(* Logix 5000 project; controller Generic 1768-L43 rev 15.6; software revision 15.01; part 10 of 10 *)
(* tags used below, declared in another part *)
   Axis_00_CMD : UDT_Axis_CMD;
   Axis_00_Data : UDT_Axis_Data;
   AXIS_01 : AXIS_SERVO_DRIVE;
   Axis_01_CMD : UDT_Axis_CMD;
   Axis_01_Data : UDT_Axis_Data;
   Axis_01_Status : UDT_Axis_Status;
   AXIS_02 : AXIS_SERVO_DRIVE;
   Axis_02_CMD : UDT_Axis_CMD;
   Axis_02_Data : UDT_Axis_Data;
   Axis_02_Status : UDT_Axis_Status;
   AXIS_03 : AXIS_SERVO_DRIVE;
   Axis_03_CMD : UDT_Axis_CMD;
   Axis_03_Data : UDT_Axis_Data;
   Axis_03_Status : UDT_Axis_Status;
   AXIS_04 : AXIS_SERVO_DRIVE;
   Axis_04_CMD : UDT_Axis_CMD;
   Axis_04_Data : UDT_Axis_Data;
   Axis_04_Status : UDT_Axis_Status;
   GenericMachine_COND : UDT_Machine_COND;
   GUI_Axis_01_JogFwdREQ : BOOL;
   GUI_Axis_01_JogRevREQ : BOOL;
   GUI_Axis_01_ReferenceREQ : BOOL;
   GUI_Axis_02_JogFwdREQ : BOOL;
   GUI_Axis_02_JogRevREQ : BOOL;
   GUI_Axis_02_ReferenceREQ : BOOL;
   GUI_Axis_03_JogFwdREQ : BOOL;
   GUI_Axis_03_JogRevREQ : BOOL;
   GUI_Axis_03_ReferenceREQ : BOOL;
   GUI_Axis_04_JogFwdREQ : BOOL;
   GUI_Axis_04_JogRevREQ : BOOL;
   GUI_Axis_04_ReferenceREQ : BOOL;
   GUI_ReferenceREQ : BOOL;
   PhaseTimout : UDT_PhaseTimeout;
   PZ_GenericMachine_AUTO : PHASE;
   PZ_GenericMachine_MANUAL : PHASE;
(* PZ_GenericMachine_AUTO, continued *)

ROUTINE Running   (* ladder *)
// CONTROLS MACHINE RUNNING PHASE.  MODIFY AS NEEDED.
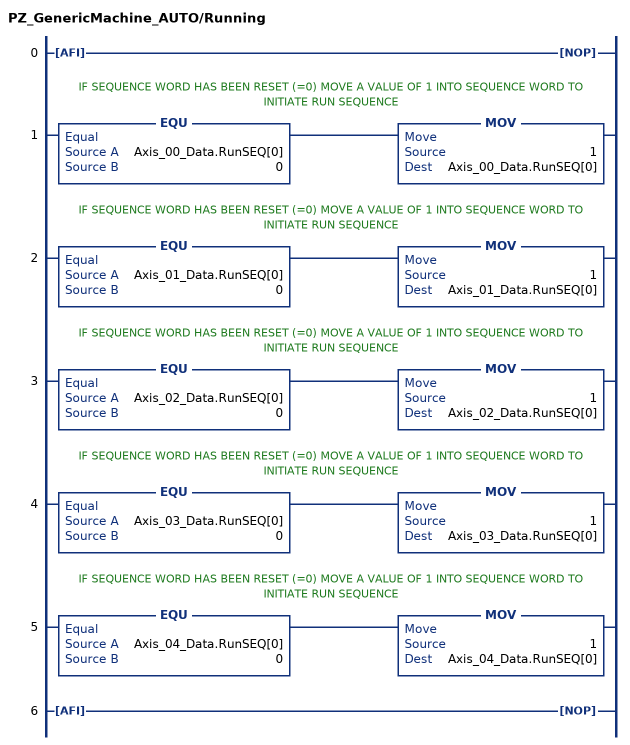
   0: AFI()NOP();
   // IF SEQUENCE WORD HAS BEEN RESET (=0) MOVE A VALUE OF 1 INTO SEQUENCE WORD TO INITIATE RUN SEQUENCE
   1: EQU(Axis_00_Data.RunSEQ[0],0)MOV(1,Axis_00_Data.RunSEQ[0]);
   // IF SEQUENCE WORD HAS BEEN RESET (=0) MOVE A VALUE OF 1 INTO SEQUENCE WORD TO INITIATE RUN SEQUENCE
   2: EQU(Axis_01_Data.RunSEQ[0],0)MOV(1,Axis_01_Data.RunSEQ[0]);
   // IF SEQUENCE WORD HAS BEEN RESET (=0) MOVE A VALUE OF 1 INTO SEQUENCE WORD TO INITIATE RUN SEQUENCE
   3: EQU(Axis_02_Data.RunSEQ[0],0)MOV(1,Axis_02_Data.RunSEQ[0]);
   // IF SEQUENCE WORD HAS BEEN RESET (=0) MOVE A VALUE OF 1 INTO SEQUENCE WORD TO INITIATE RUN SEQUENCE
   4: EQU(Axis_03_Data.RunSEQ[0],0)MOV(1,Axis_03_Data.RunSEQ[0]);
   // IF SEQUENCE WORD HAS BEEN RESET (=0) MOVE A VALUE OF 1 INTO SEQUENCE WORD TO INITIATE RUN SEQUENCE
   5: EQU(Axis_04_Data.RunSEQ[0],0)MOV(1,Axis_04_Data.RunSEQ[0]);
   6: AFI()NOP();
END_ROUTINE

ROUTINE Stopping   (* ladder *)
// CONTROLS MACHINE STOPPING PHASE.  MODIFY AS NEEDED.
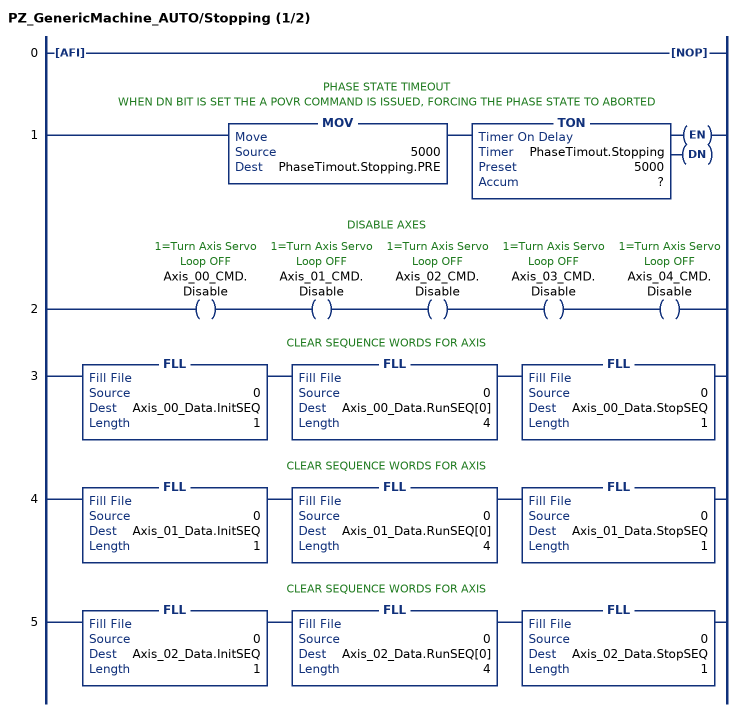
   0: AFI()NOP();
   // PHASE STATE TIMEOUT
   //   WHEN DN BIT IS SET THE A POVR COMMAND IS ISSUED, FORCING THE PHASE STATE TO ABORTED
   1: MOV(5000,PhaseTimout.Stopping.PRE)TON(PhaseTimout.Stopping,?,?);
   // DISABLE AXES
   2: OTE(Axis_00_CMD.Disable)OTE(Axis_01_CMD.Disable)OTE(Axis_02_CMD.Disable)OTE(Axis_03_CMD.Disable)OTE(Axis_04_CMD.Disable);
   // CLEAR SEQUENCE WORDS FOR AXIS
   3: FLL(0,Axis_00_Data.InitSEQ,1)FLL(0,Axis_00_Data.RunSEQ[0],4)FLL(0,Axis_00_Data.StopSEQ,1);
   // CLEAR SEQUENCE WORDS FOR AXIS
   4: FLL(0,Axis_01_Data.InitSEQ,1)FLL(0,Axis_01_Data.RunSEQ[0],4)FLL(0,Axis_01_Data.StopSEQ,1);
   // CLEAR SEQUENCE WORDS FOR AXIS
   5: FLL(0,Axis_02_Data.InitSEQ,1)FLL(0,Axis_02_Data.RunSEQ[0],4)FLL(0,Axis_02_Data.StopSEQ,1);
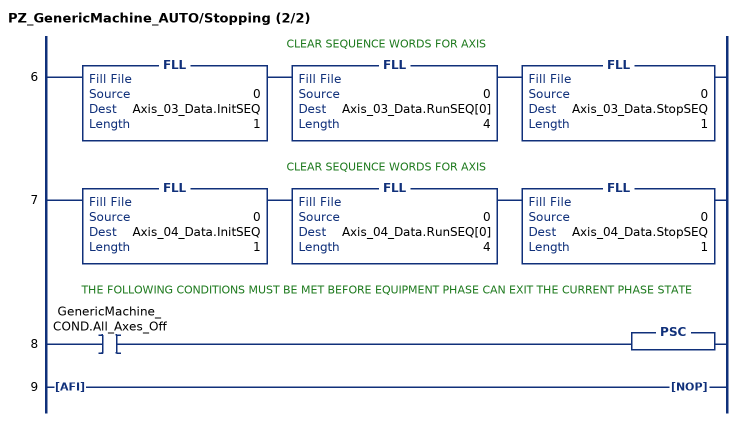
   // CLEAR SEQUENCE WORDS FOR AXIS
   6: FLL(0,Axis_03_Data.InitSEQ,1)FLL(0,Axis_03_Data.RunSEQ[0],4)FLL(0,Axis_03_Data.StopSEQ,1);
   // CLEAR SEQUENCE WORDS FOR AXIS
   7: FLL(0,Axis_04_Data.InitSEQ,1)FLL(0,Axis_04_Data.RunSEQ[0],4)FLL(0,Axis_04_Data.StopSEQ,1);
   // THE FOLLOWING CONDITIONS MUST BE MET BEFORE EQUIPMENT PHASE CAN EXIT THE CURRENT PHASE STATE
   8: XIC(GenericMachine_COND.All_Axes_Off)PSC();
   9: AFI()NOP();
END_ROUTINE
END_PROGRAM

PROGRAM PZ_GenericMachine_MANUAL

ROUTINE Aborting   (* ladder *)
// CONTROLS MACHINE MANUAL ABORTING PHASE.  MODIFY AS NEEDED.
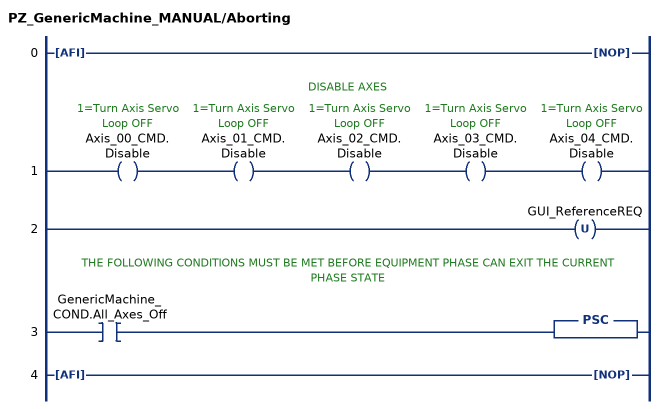
   0: AFI()NOP();
   // DISABLE AXES
   1: OTE(Axis_00_CMD.Disable)OTE(Axis_01_CMD.Disable)OTE(Axis_02_CMD.Disable)OTE(Axis_03_CMD.Disable)OTE(Axis_04_CMD.Disable);
   2: OTU(GUI_ReferenceREQ);
   // THE FOLLOWING CONDITIONS MUST BE MET BEFORE EQUIPMENT PHASE CAN EXIT THE CURRENT PHASE STATE
   3: XIC(GenericMachine_COND.All_Axes_Off)PSC();
   4: AFI()NOP();
END_ROUTINE

ROUTINE Resetting   (* ladder *)
// CONTROLS MACHINE MANUAL RESETTING PHASE.  MODIFY AS NEEDED.
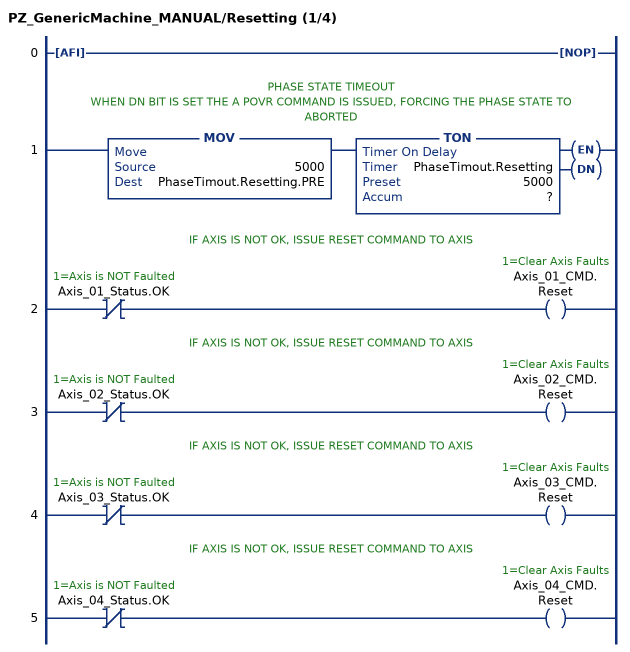
   0: AFI()NOP();
   // PHASE STATE TIMEOUT
   //   WHEN DN BIT IS SET THE A POVR COMMAND IS ISSUED, FORCING THE PHASE STATE TO ABORTED
   1: MOV(5000,PhaseTimout.Resetting.PRE)TON(PhaseTimout.Resetting,?,?);
   // IF AXIS IS NOT OK, ISSUE RESET COMMAND TO AXIS
   2: XIO(Axis_01_Status.OK)OTE(Axis_01_CMD.Reset);
   // IF AXIS IS NOT OK, ISSUE RESET COMMAND TO AXIS
   3: XIO(Axis_02_Status.OK)OTE(Axis_02_CMD.Reset);
   // IF AXIS IS NOT OK, ISSUE RESET COMMAND TO AXIS
   4: XIO(Axis_03_Status.OK)OTE(Axis_03_CMD.Reset);
   // IF AXIS IS NOT OK, ISSUE RESET COMMAND TO AXIS
   5: XIO(Axis_04_Status.OK)OTE(Axis_04_CMD.Reset);
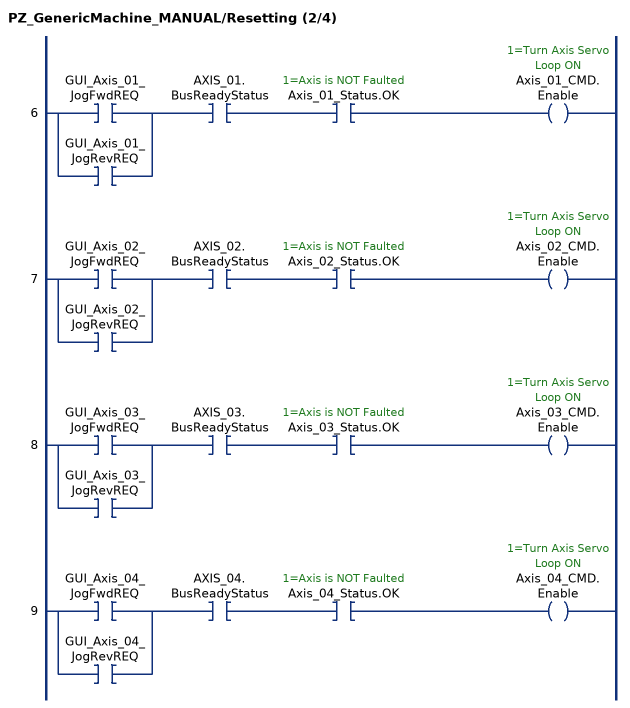
   6: [XIC(GUI_Axis_01_JogFwdREQ) ,XIC(GUI_Axis_01_JogRevREQ) ]XIC(AXIS_01.BusReadyStatus)XIC(Axis_01_Status.OK)OTE(Axis_01_CMD.Enable);
   7: [XIC(GUI_Axis_02_JogFwdREQ) ,XIC(GUI_Axis_02_JogRevREQ) ]XIC(AXIS_02.BusReadyStatus)XIC(Axis_02_Status.OK)OTE(Axis_02_CMD.Enable);
   8: [XIC(GUI_Axis_03_JogFwdREQ) ,XIC(GUI_Axis_03_JogRevREQ) ]XIC(AXIS_03.BusReadyStatus)XIC(Axis_03_Status.OK)OTE(Axis_03_CMD.Enable);
   9: [XIC(GUI_Axis_04_JogFwdREQ) ,XIC(GUI_Axis_04_JogRevREQ) ]XIC(AXIS_04.BusReadyStatus)XIC(Axis_04_Status.OK)OTE(Axis_04_CMD.Enable);
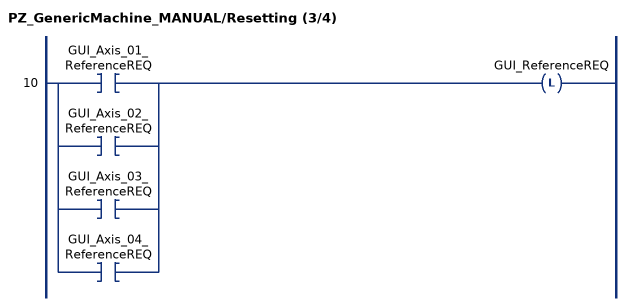
   10: [XIC(GUI_Axis_01_ReferenceREQ) ,XIC(GUI_Axis_02_ReferenceREQ) ,XIC(GUI_Axis_03_ReferenceREQ) ,XIC(GUI_Axis_04_ReferenceREQ) ]OTL(GUI_ReferenceREQ);
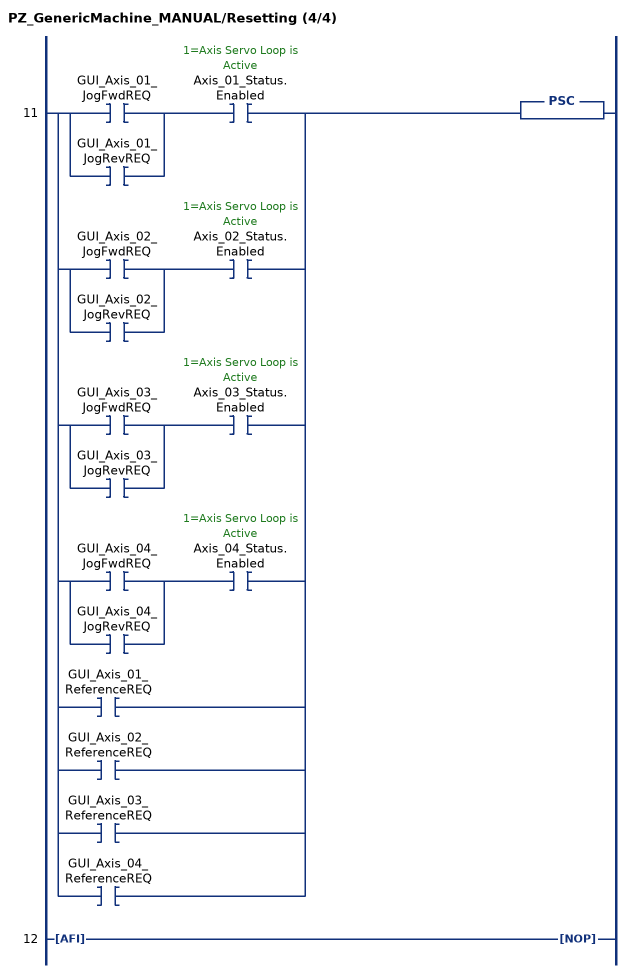
   11: [[XIC(GUI_Axis_01_JogFwdREQ) ,XIC(GUI_Axis_01_JogRevREQ) ] XIC(Axis_01_Status.Enabled) ,[XIC(GUI_Axis_02_JogFwdREQ) ,XIC(GUI_Axis_02_JogRevREQ) ] XIC(Axis_02_Status.Enabled) ,[XIC(GUI_Axis_03_JogFwdREQ) ,XIC(GUI_Axis_03_JogRevREQ) ] XIC(Axis_03_Status.Enabled) ,[XIC(GUI_Axis_04_JogFwdREQ) ,XIC(GUI_Axis_04_JogRevREQ) ] XIC(Axis_04_Status.Enabled) ,XIC(GUI_Axis_01_ReferenceREQ) ,XIC(GUI_Axis_02_ReferenceREQ) ,XIC(GUI_Axis_03_ReferenceREQ) ,XIC(GUI_Axis_04_ReferenceREQ) ]PSC();
   12: AFI()NOP();
END_ROUTINE

ROUTINE Running   (* ladder *)
// CONTROLS MACHINE MANUAL RUNNING PHASE.  MODIFY AS NEEDED.
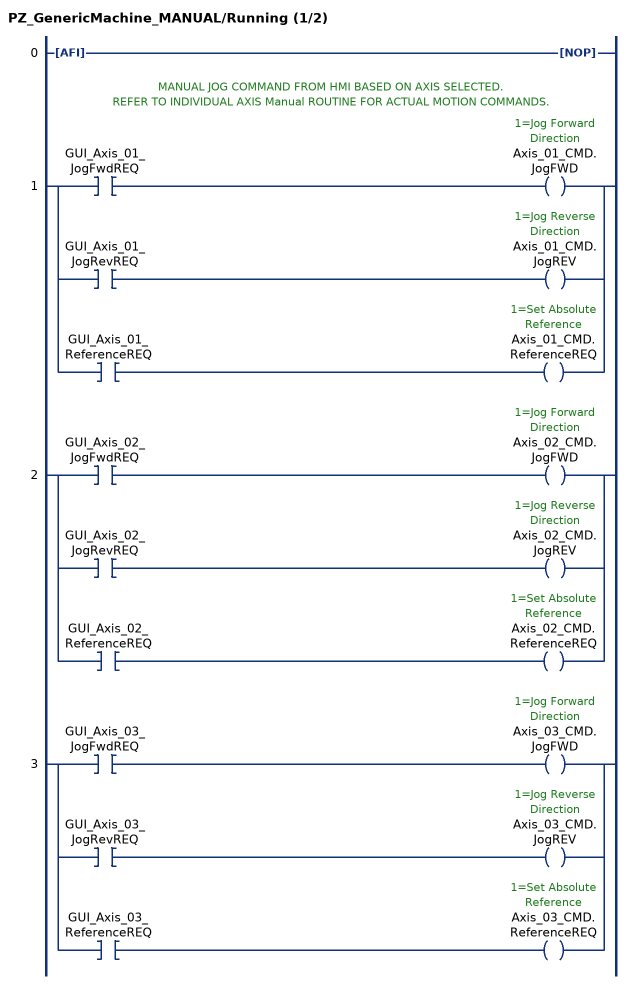
   0: AFI()NOP();
   // MANUAL JOG COMMAND FROM HMI BASED ON AXIS SELECTED.
   // REFER TO INDIVIDUAL AXIS Manual ROUTINE FOR ACTUAL MOTION COMMANDS.
   1: [XIC(GUI_Axis_01_JogFwdREQ) OTE(Axis_01_CMD.JogFWD) ,XIC(GUI_Axis_01_JogRevREQ) OTE(Axis_01_CMD.JogREV) ,XIC(GUI_Axis_01_ReferenceREQ) OTE(Axis_01_CMD.ReferenceREQ) ];
   2: [XIC(GUI_Axis_02_JogFwdREQ) OTE(Axis_02_CMD.JogFWD) ,XIC(GUI_Axis_02_JogRevREQ) OTE(Axis_02_CMD.JogREV) ,XIC(GUI_Axis_02_ReferenceREQ) OTE(Axis_02_CMD.ReferenceREQ) ];
   3: [XIC(GUI_Axis_03_JogFwdREQ) OTE(Axis_03_CMD.JogFWD) ,XIC(GUI_Axis_03_JogRevREQ) OTE(Axis_03_CMD.JogREV) ,XIC(GUI_Axis_03_ReferenceREQ) OTE(Axis_03_CMD.ReferenceREQ) ];
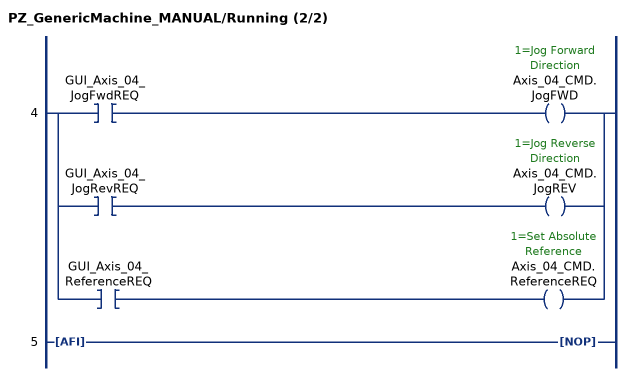
   4: [XIC(GUI_Axis_04_JogFwdREQ) OTE(Axis_04_CMD.JogFWD) ,XIC(GUI_Axis_04_JogRevREQ) OTE(Axis_04_CMD.JogREV) ,XIC(GUI_Axis_04_ReferenceREQ) OTE(Axis_04_CMD.ReferenceREQ) ];
   5: AFI()NOP();
END_ROUTINE

ROUTINE Stopping   (* ladder *)
// CONTROLS MACHINE MANUAL STOPPING PHASE.  MODIFY AS NEEDED.
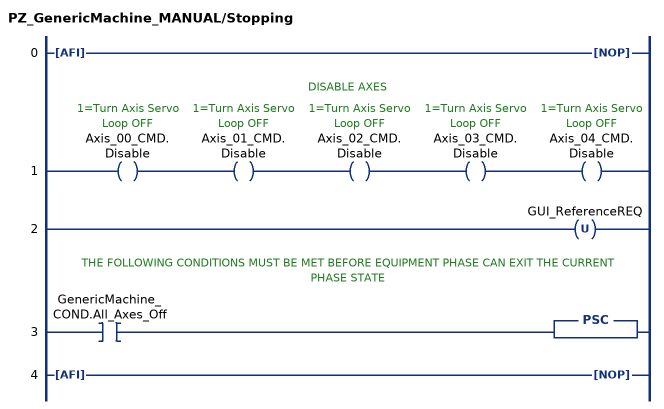
   0: AFI()NOP();
   // DISABLE AXES
   1: OTE(Axis_00_CMD.Disable)OTE(Axis_01_CMD.Disable)OTE(Axis_02_CMD.Disable)OTE(Axis_03_CMD.Disable)OTE(Axis_04_CMD.Disable);
   2: OTU(GUI_ReferenceREQ);
   // THE FOLLOWING CONDITIONS MUST BE MET BEFORE EQUIPMENT PHASE CAN EXIT THE CURRENT PHASE STATE
   3: XIC(GenericMachine_COND.All_Axes_Off)PSC();
   4: AFI()NOP();
END_ROUTINE
END_PROGRAM
